FUNCTION_BLOCK controller_p
VAR_INPUT
	b_start: BOOL;
	t_time: TIME;
END_VAR		
VAR_OUTPUT
	x_trigger: BOOL;
END_VAR
VAR
	fb_Pulse1: TP;
	fb_Pulse2: TP;
	fb_ftrig1: F_TRIG;
	fb_ftrig2: F_TRIG;
	b_StartTimer1: BOOL;
	b_StartTimer2: BOOL;
END_VAR

IF b_start THEN
	fb_Pulse1(IN:=b_StartTimer1,PT:=t_time);
	fb_Pulse2(IN:=b_StartTimer2,PT:=t_time);
	
	fb_ftrig1.CLK:= fb_Pulse1.Q;
	fb_ftrig2.CLK:= fb_Pulse2.Q;
	
	IF NOT fb_Pulse1.Q AND NOT fb_Pulse2.Q THEN
		b_StartTimer1:= TRUE;
		b_StartTimer2:= FALSE;
		
	ELSIF fb_ftrig1.Q THEN
		b_StartTimer1:= FALSE;
		b_StartTimer2:= TRUE;
		
	ELSIF fb_ftrig2.Q THEN
		b_StartTimer1:= TRUE;
		b_StartTimer2:= FALSE;
	END_IF
	
ELSE
	b_StartTimer1:= FALSE;
	b_StartTimer2:= FALSE;
	x_trigger:= FALSE;
END_IF

END_FUNCTION_BLOCK

(* stored: Version 1.1.0.1, ProductVersion 3.1.4022.7
   POU controller_p: Id {749bdadd-d2e5-4dc7-ab57-4c0ea94e0d9c}, SpecialFunc None *)
